// TIA Portal V18 export
DATA_BLOCK "RPM"   // DB77
{ S7_Optimized_Access := 'TRUE' }
VERSION : 0.1
// stored: AutoNumber true, DBAccessibleFromOPCUA true, IsOnlyStoredInLoadMemory false, IsRetainMemResEnabled false, IsWriteProtectedInAS false, MemoryReserve 100
   VAR
      "A" : Real;
      "B" : Real;
   END_VAR
   VAR RETAIN
      "speed sensor selection A" : Int;
      "speed sensor selection B" : Int;
   END_VAR
   VAR
      "a selected" : Bool;
      "b selected" : Bool;
      "ab selected" : Bool;
      "No signal RPM sensor A" : Bool;
      "No signal RPM sensor B" : Bool;
      "A frequency" : Real;
      "B frequency" : Real;
   END_VAR
BEGIN
END_DATA_BLOCK
